INTERFACE INTERNAL _I_Worker EXTENDS I_Debug, I_ValidateInterface;

PROPERTY INTERNAL _Next : I_Worker
GET
END_GET
SET
END_SET
END_PROPERTY

PROPERTY INTERNAL _Prev : I_Worker
GET
END_GET
SET
END_SET
END_PROPERTY

PROPERTY INTERNAL _PlantNext : I_Worker
GET
END_GET
SET
END_SET
END_PROPERTY

PROPERTY INTERNAL _PlantPrev : I_Worker
GET
END_GET
SET
END_SET
END_PROPERTY

METHOD INTERNAL Process
VAR_OUTPUT
	iNext: I_Worker;
END_VAR
END_METHOD

PROPERTY INTERNAL _Thread : I_Thread
GET
END_GET
SET
END_SET
END_PROPERTY

// Thread that processes this worker; can change while Idle.
PROPERTY Thread : I_Thread
GET
END_GET
SET
END_SET
END_PROPERTY

END_INTERFACE

(* stored: Version 1.1.0.1
   Itf _I_Worker: Id {07430000-e899-49ca-9847-972737ca3f53}
   Property _Next: Id {426096a7-01e2-40c8-a7dd-d67bd6f6a327}
   Get Get: Id {ec3f1859-9bac-4254-a57c-9db6e7eb29cf}
   Set Set: Id {677614c4-5f73-475a-b54d-cb7b12bb9a90}
   Property _Prev: Id {db271ff8-3568-4693-8384-2665bec344a9}
   Get Get: Id {b65827bb-4606-4fd8-8596-4b34ee1291ea}
   Set Set: Id {ccd5eece-c562-41e4-903f-9e6dcacf894d}
   Property _PlantNext: Id {c6d58d7a-2cd6-4afd-8daa-ed94a0208514}
   Get Get: Id {3d896fcf-8d59-42a3-967a-a8e5550e2a6e}
   Set Set: Id {fb9dde27-4f2d-4d7e-b0fc-37e2334fd385}
   Property _PlantPrev: Id {0fd0ef65-3e59-4581-ae7d-feb5ba434f7f}
   Get Get: Id {923b7a69-b545-4bc4-ac5a-11803d2fedcd}
   Set Set: Id {5c50dd8f-b4c6-488d-9ce8-05dfcb3e27cd}
   Method Process: Id {bf44a028-9259-46a3-b6eb-6c366a7704c7}
   Property _Thread: Id {3aa35d64-97c9-4d18-ac1c-6f33e1ac0b2d}
   Get Get: Id {cbd7efab-dfc6-425b-bccb-3b57d4ea6d14}
   Set Set: Id {bf4380d8-eeac-4286-9690-d2db8e6d960d}
   Property Thread: Id {72664e5a-4e4f-4a16-a656-7b32bc2b89e7}
   Get Get: Id {1ae9c584-ea6d-4c91-be59-16d88dfc59d3}
   Set Set: Id {f042ba81-7885-4cd1-8f03-fcb05f790817} *)
